Staubli VAL3: start.pgx

program start()
begin

  // read file
  call util:readFile("Disk://input_day1.txt", sInput)

  // PUZZLE 1
  // vec2num
  call util:vec2num(sInput, nInput)

  // calc diff between elements
  call math:diff(nInput, nResult2)

  // compare elements if step is >0
  call util:compare(nResult2, ">", 0, bResult)

  // count steps > 0
  call util:countBool(bResult, nResult)
  ? nResult

  // PUZZLE 2
  call math:rollsum(nInput, 3, nResult)

  // calc diff between elements
  call math:diff(nResult, nResult2)

  // compare elements if step is >0
  call util:compare(nResult2, ">", 0, bResult)

  // count steps > 0
  call util:countBool(bResult, nResult)
  ? nResult

end
